TYPE Taak_2 :
	(
		functie,
		Inladen,
		Transport,
		Afleveren,
		Retour
	) := Inladen;
END_TYPE

(* stored: Version 1.1.0.1, ProductVersion 3.1.4024.12
   DUT Taak_2: Id {5a82a080-f46b-4cfc-a059-90891e7b3d47} *)
